# EPICS substitutions: modules/ip330/ip330App/Db/IP330.substitutions
#==============================================================================
#
# Abs:  Acromag IP-330 ADC template
#
# Name: IP330.substitutions
#
#  Auth: 10-Aug-2006, S. Peng         (PENG)
#  Rev:  dd-mmm-yyyy, Reviewer's Name (USERNAME)
#-----------------------------------------------------------------------------
# Mod:
#       dd-mmm-yyyy, First lastname (USERNAME):
#         comment
#
#==============================================================================
#
file IP330.template
{
  pattern { RECNAME,                CARD  ,  CH,  EFUG,  EGUL, ADEL,  MDEL, HIHI,  HIGH, LOW , LOLO,  EGU   }
          { LCLS:IP_TEST:AI:C$(CH), "ai0" ,   0,  5.0 ,  0.0 , 0.0 ,  0.0 , 4.5 ,  4.0 , 1.0 , 0.5 ,  Volts }
          { LCLS:IP_TEST:AI:C$(CH), "ai0" ,   1,  5.0 ,  0.0 , 0.0 ,  0.0 , 4.5 ,  4.0 , 1.0 , 0.5 ,  Volts }
          { LCLS:IP_TEST:AI:C$(CH), "ai0" ,   2,  5.0 ,  0.0 , 0.0 ,  0.0 , 4.5 ,  4.0 , 1.0 , 0.5 ,  Volts }
          { LCLS:IP_TEST:AI:C$(CH), "ai0" ,   3,  5.0 ,  0.0 , 0.0 ,  0.0 , 4.5 ,  4.0 , 1.0 , 0.5 ,  Volts }
          { LCLS:IP_TEST:AI:C$(CH), "ai0" ,   4,  5.0 ,  0.0 , 0.0 ,  0.0 , 4.5 ,  4.0 , 1.0 , 0.5 ,  Volts }
          { LCLS:IP_TEST:AI:C$(CH), "ai0" ,   5,  5.0 ,  0.0 , 0.0 ,  0.0 , 4.5 ,  4.0 , 1.0 , 0.5 ,  Volts }
          { LCLS:IP_TEST:AI:C$(CH), "ai0" ,   6,  5.0 ,  0.0 , 0.0 ,  0.0 , 4.5 ,  4.0 , 1.0 , 0.5 ,  Volts }
          { LCLS:IP_TEST:AI:C$(CH), "ai0" ,   7,  5.0 ,  0.0 , 0.0 ,  0.0 , 4.5 ,  4.0 , 1.0 , 0.5 ,  Volts }
          { LCLS:IP_TEST:AI:C$(CH), "ai0" ,   8,  5.0 ,  0.0 , 0.0 ,  0.0 , 4.5 ,  4.0 , 1.0 , 0.5 ,  Volts }
          { LCLS:IP_TEST:AI:C$(CH), "ai0" ,   9,  5.0 ,  0.0 , 0.0 ,  0.0 , 4.5 ,  4.0 , 1.0 , 0.5 ,  Volts }
          { LCLS:IP_TEST:AI:C$(CH), "ai0" ,  10,  5.0 ,  0.0 , 0.0 ,  0.0 , 4.5 ,  4.0 , 1.0 , 0.5 ,  Volts }
          { LCLS:IP_TEST:AI:C$(CH), "ai0" ,  11,  5.0 ,  0.0 , 0.0 ,  0.0 , 4.5 ,  4.0 , 1.0 , 0.5 ,  Volts }
          { LCLS:IP_TEST:AI:C$(CH), "ai0" ,  12,  5.0 ,  0.0 , 0.0 ,  0.0 , 4.5 ,  4.0 , 1.0 , 0.5 ,  Volts }
          { LCLS:IP_TEST:AI:C$(CH), "ai0" ,  13,  5.0 ,  0.0 , 0.0 ,  0.0 , 4.5 ,  4.0 , 1.0 , 0.5 ,  Volts }
          { LCLS:IP_TEST:AI:C$(CH), "ai0" ,  14,  5.0 ,  0.0 , 0.0 ,  0.0 , 4.5 ,  4.0 , 1.0 , 0.5 ,  Volts }
          { LCLS:IP_TEST:AI:C$(CH), "ai0" ,  15,  5.0 ,  0.0 , 0.0 ,  0.0 , 4.5 ,  4.0 , 1.0 , 0.5 ,  Volts }
}
